FUNCTION_BLOCK InputSender (* Composite Function Block Type *)
  (* Standard: 61499-2 *)
  (* Version 0.0, 6/20/2018, Rediska, nxtControl GmbH, template *)
  PACKAGE Main;
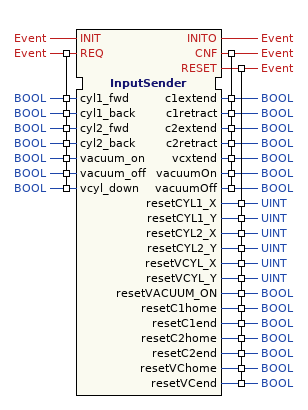
  EVENT_INPUT
    INIT; (* Initialization Request *)
    REQ WITH cyl1_fwd, cyl1_back, cyl2_fwd, cyl2_back, vacuum_on, vacuum_off, vcyl_down; (* Normal Execution Request *)
  END_EVENT
  EVENT_OUTPUT
    INITO; (* Initialization Confirm *)
    CNF WITH c1extend, c1retract, c2extend, c2retract, vcxtend, vacuumOn, vacuumOff; (* Execution Confirmation *)
    RESET WITH resetCYL1_X, resetCYL1_Y, resetCYL2_X, resetCYL2_Y, resetVCYL_X, resetVCYL_Y, resetVACUUM_ON, resetC1home, resetC1end, resetC2home, resetC2end, resetVChome, resetVCend;
  END_EVENT
  VAR_INPUT
    cyl1_fwd : BOOL;
    cyl1_back : BOOL;
    cyl2_fwd : BOOL;
    cyl2_back : BOOL;
    vacuum_on : BOOL;
    vacuum_off : BOOL;
    vcyl_down : BOOL;
  END_VAR
  VAR_OUTPUT
    c1extend : BOOL;
    c1retract : BOOL;
    c2extend : BOOL;
    c2retract : BOOL;
    vcxtend : BOOL;
    vacuumOn : BOOL;
    vacuumOff : BOOL;
    resetCYL1_X : UINT;
    resetCYL1_Y : UINT;
    resetCYL2_X : UINT;
    resetCYL2_Y : UINT;
    resetVCYL_X : UINT;
    resetVCYL_Y : UINT;
    resetVACUUM_ON : BOOL;
    resetC1home : BOOL;
    resetC1end : BOOL;
    resetC2home : BOOL;
    resetC2end : BOOL;
    resetVChome : BOOL;
    resetVCend : BOOL;
  END_VAR
  FBS
    FB2 : TCPIO(PORT := ;127.0.0.1:64999);
    FB3 : InputDecompressor(delimiter := ;);
    FB1 : InputCompressor(delimiter := ;);
  END_FBS
  EVENT_CONNECTIONS
    INIT TO FB1.INIT;
    REQ TO FB1.REQ;
    FB3.INITO TO INITO;
    FB3.CNF TO CNF;
    FB1.INITO TO FB2.INIT;
    FB1.CNF TO FB2.REQ;
    FB2.CNF TO FB2.ACK;
    FB2.INITO TO FB3.INIT;
    FB2.IND TO FB3.REQ;
    FB3.RESET TO RESET;
  END_CONNECTIONS
  DATA_CONNECTIONS
    cyl1_fwd TO FB1.cyl1_fwd;
    cyl1_back TO FB1.cyl1_back;
    cyl2_fwd TO FB1.cyl2_fwd;
    cyl2_back TO FB1.cyl2_back;
    vacuum_on TO FB1.vacuum_on;
    vacuum_off TO FB1.vacuum_off;
    vcyl_down TO FB1.vcyl_down;
    FB1.RESULT TO FB2.DATAOUT;
    FB1.QO TO FB2.QI;
    FB2.QO TO FB3.QI;
    FB2.DATAIN TO FB3.input;
    FB3.cyl1_back TO c1retract;
    FB3.cyl2_fwd TO c2extend;
    FB3.cyl2_back TO c2retract;
    FB3.vcyl_down TO vcxtend;
    FB3.vacuum_on TO vacuumOn;
    FB3.vacuum_off TO vacuumOff;
    FB3.resetCYL1_X TO resetCYL1_X;
    FB3.resetCYL1_Y TO resetCYL1_Y;
    FB3.resetCYL2_X TO resetCYL2_X;
    FB3.resetCYL2_Y TO resetCYL2_Y;
    FB3.resetVCYL_X TO resetVCYL_X;
    FB3.resetVCYL_Y TO resetVCYL_Y;
    FB3.resetVACUUM_ON TO resetVACUUM_ON;
    FB3.resetC1home TO resetC1home;
    FB3.resetC1end TO resetC1end;
    FB3.resetC2home TO resetC2home;
    FB3.resetC2end TO resetC2end;
    FB3.resetVchome TO resetVChome;
    FB3.resetVcend TO resetVCend;
  END_CONNECTIONS
END_FUNCTION_BLOCK
